// TIA Portal V18 program export: 0 tag tables, 0 data types, 0 data blocks, 2 code blocks (in call order from the OBs), 6 instance data blocks

ORGANIZATION_BLOCK "Main"   // OB1, LAD, ProgramCycle
TITLE = "Main Program Sweep (Cycle)"
{ S7_Optimized_Access := 'TRUE' }
VERSION : 0.1
// Este bloco verifica as condições dos sinais discretos dos painéis. Se as condições operacionais não forem atendidas, as FCs respectivas de cada painel são intertravadas no item 2. Fluxo de Controle.
// stored: AutoNumber true, IsIECCheckEnabled false, SetENOAutomatically false
   VAR_INPUT
      Initial_Call : Bool;   // Initial call of this OB
      Remanence : Bool;   // =True, if remanent data are available
   END_VAR
BEGIN

REGION Network 1: Intertravamento Painel CCO
   // Se o Botão de Emergência estiver Desacionado Painel CCO OK
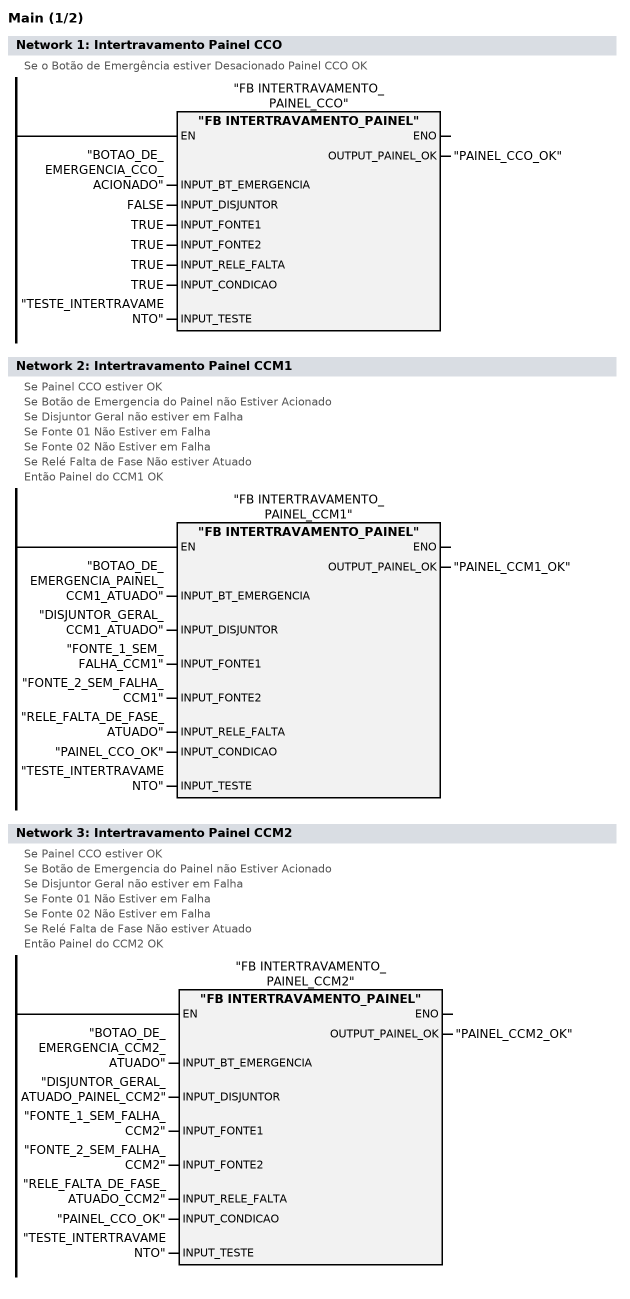
   RUNG wire#powerrail
      "FB INTERTRAVAMENTO_PAINEL_CCO"(INPUT_BT_EMERGENCIA := "BOTAO_DE_EMERGENCIA_CCO_ACIONADO", INPUT_DISJUNTOR := FALSE, INPUT_FONTE1 := TRUE, INPUT_FONTE2 := TRUE, INPUT_RELE_FALTA := TRUE, INPUT_CONDICAO := TRUE, INPUT_TESTE := "TESTE_INTERTRAVAMENTO", OUTPUT_PAINEL_OK => "PAINEL_CCO_OK")
   END_RUNG
   // the same network as SCL:
   "FB INTERTRAVAMENTO_PAINEL_CCO"(INPUT_BT_EMERGENCIA := "BOTAO_DE_EMERGENCIA_CCO_ACIONADO",   // "FB INTERTRAVAMENTO_PAINEL"
                           INPUT_DISJUNTOR := FALSE,
                           INPUT_FONTE1 := TRUE,
                           INPUT_FONTE2 := TRUE,
                           INPUT_RELE_FALTA := TRUE,
                           INPUT_CONDICAO := TRUE,
                           INPUT_TESTE := "TESTE_INTERTRAVAMENTO",
                           OUTPUT_PAINEL_OK => "PAINEL_CCO_OK");
END_REGION

REGION Network 2: Intertravamento Painel CCM1
   // Se Painel CCO estiver OK
   // Se Botão de Emergencia do Painel não Estiver Acionado
   // Se Disjuntor Geral não estiver em Falha
   // Se Fonte 01 Não Estiver em Falha
   // Se Fonte 02 Não Estiver em Falha
   // Se Relé Falta de Fase Não estiver Atuado
   // Então Painel do CCM1 OK
   RUNG wire#powerrail
      "FB INTERTRAVAMENTO_PAINEL_CCM1"(INPUT_BT_EMERGENCIA := "BOTAO_DE_EMERGENCIA_PAINEL_CCM1_ATUADO", INPUT_DISJUNTOR := "DISJUNTOR_GERAL_CCM1_ATUADO", INPUT_FONTE1 := "FONTE_1_SEM_ FALHA_CCM1", INPUT_FONTE2 := "FONTE_2_SEM_FALHA_CCM1", INPUT_RELE_FALTA := "RELE_FALTA_DE_FASE_ATUADO", INPUT_CONDICAO := "PAINEL_CCO_OK", INPUT_TESTE := "TESTE_INTERTRAVAMENTO", OUTPUT_PAINEL_OK => "PAINEL_CCM1_OK")
   END_RUNG
   // the same network as SCL:
   "FB INTERTRAVAMENTO_PAINEL_CCM1"(INPUT_BT_EMERGENCIA := "BOTAO_DE_EMERGENCIA_PAINEL_CCM1_ATUADO",   // "FB INTERTRAVAMENTO_PAINEL"
                           INPUT_DISJUNTOR := "DISJUNTOR_GERAL_CCM1_ATUADO",
                           INPUT_FONTE1 := "FONTE_1_SEM_ FALHA_CCM1",
                           INPUT_FONTE2 := "FONTE_2_SEM_FALHA_CCM1",
                           INPUT_RELE_FALTA := "RELE_FALTA_DE_FASE_ATUADO",
                           INPUT_CONDICAO := "PAINEL_CCO_OK",
                           INPUT_TESTE := "TESTE_INTERTRAVAMENTO",
                           OUTPUT_PAINEL_OK => "PAINEL_CCM1_OK");
END_REGION

REGION Network 3: Intertravamento Painel CCM2
   // Se Painel CCO estiver OK
   // Se Botão de Emergencia do Painel não Estiver Acionado
   // Se Disjuntor Geral não estiver em Falha
   // Se Fonte 01 Não Estiver em Falha
   // Se Fonte 02 Não Estiver em Falha
   // Se Relé Falta de Fase Não estiver Atuado
   // Então Painel do CCM2 OK
   RUNG wire#powerrail
      "FB INTERTRAVAMENTO_PAINEL_CCM2"(INPUT_BT_EMERGENCIA := "BOTAO_DE_EMERGENCIA_CCM2_ATUADO", INPUT_DISJUNTOR := "DISJUNTOR_GERAL_ATUADO_PAINEL_CCM2", INPUT_FONTE1 := "FONTE_1_SEM_FALHA_CCM2", INPUT_FONTE2 := "FONTE_2_SEM_FALHA_CCM2", INPUT_RELE_FALTA := "RELE_FALTA_DE_FASE_ATUADO_CCM2", INPUT_CONDICAO := "PAINEL_CCO_OK", INPUT_TESTE := "TESTE_INTERTRAVAMENTO", OUTPUT_PAINEL_OK => "PAINEL_CCM2_OK")
   END_RUNG
   // the same network as SCL:
   "FB INTERTRAVAMENTO_PAINEL_CCM2"(INPUT_BT_EMERGENCIA := "BOTAO_DE_EMERGENCIA_CCM2_ATUADO",   // "FB INTERTRAVAMENTO_PAINEL"
                           INPUT_DISJUNTOR := "DISJUNTOR_GERAL_ATUADO_PAINEL_CCM2",
                           INPUT_FONTE1 := "FONTE_1_SEM_FALHA_CCM2",
                           INPUT_FONTE2 := "FONTE_2_SEM_FALHA_CCM2",
                           INPUT_RELE_FALTA := "RELE_FALTA_DE_FASE_ATUADO_CCM2",
                           INPUT_CONDICAO := "PAINEL_CCO_OK",
                           INPUT_TESTE := "TESTE_INTERTRAVAMENTO",
                           OUTPUT_PAINEL_OK => "PAINEL_CCM2_OK");
END_REGION

REGION Network 4: Intertravamento Painel CCM3
   // Se Painel CCO estiver OK
   // Se Botão de Emergencia do Painel não Estiver Acionado
   // Se Disjuntor Geral não estiver em Falha
   // Se Fonte 01 Não Estiver em Falha
   // Se Fonte 02 Não Estiver em Falha
   // Se Relé Falta de Fase Não estiver Atuado
   // Então Painel do CCM1 OK
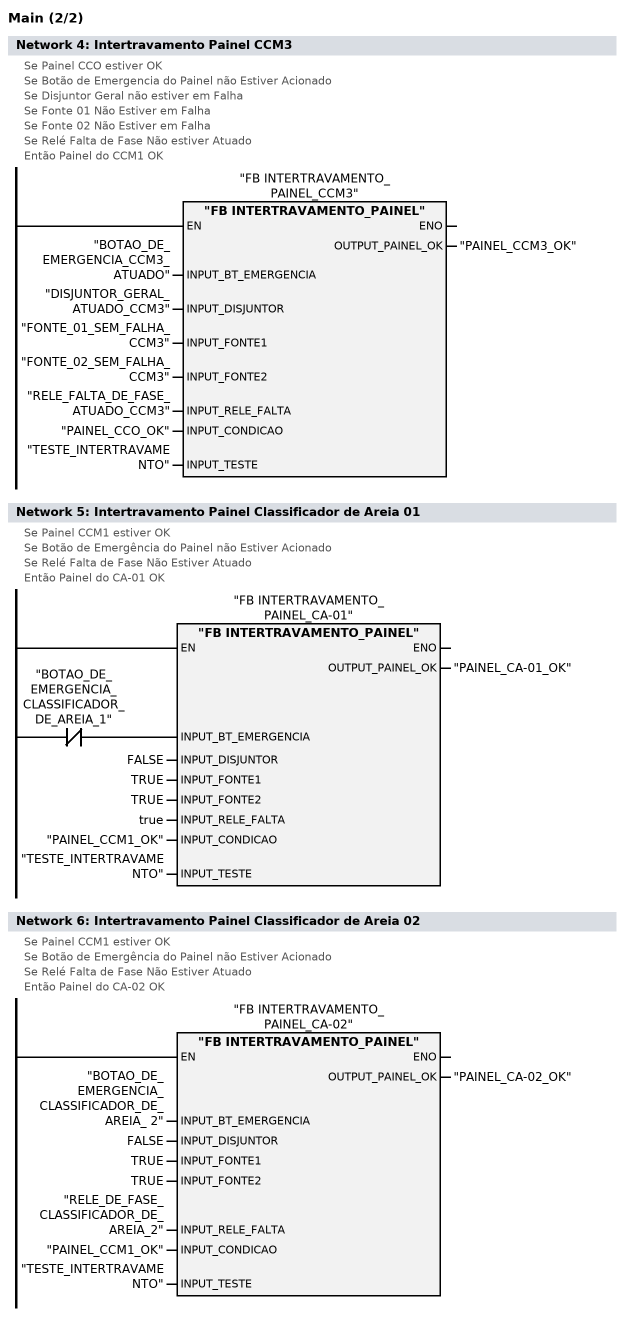
   RUNG wire#powerrail
      "FB INTERTRAVAMENTO_PAINEL_CCM3"(INPUT_BT_EMERGENCIA := "BOTAO_DE_EMERGENCIA_CCM3_ATUADO", INPUT_DISJUNTOR := "DISJUNTOR_GERAL_ATUADO_CCM3", INPUT_FONTE1 := "FONTE_01_SEM_FALHA_CCM3", INPUT_FONTE2 := "FONTE_02_SEM_FALHA_CCM3", INPUT_RELE_FALTA := "RELE_FALTA_DE_FASE_ATUADO_CCM3", INPUT_CONDICAO := "PAINEL_CCO_OK", INPUT_TESTE := "TESTE_INTERTRAVAMENTO", OUTPUT_PAINEL_OK => "PAINEL_CCM3_OK")
   END_RUNG
   // the same network as SCL:
   "FB INTERTRAVAMENTO_PAINEL_CCM3"(INPUT_BT_EMERGENCIA := "BOTAO_DE_EMERGENCIA_CCM3_ATUADO",   // "FB INTERTRAVAMENTO_PAINEL"
                           INPUT_DISJUNTOR := "DISJUNTOR_GERAL_ATUADO_CCM3",
                           INPUT_FONTE1 := "FONTE_01_SEM_FALHA_CCM3",
                           INPUT_FONTE2 := "FONTE_02_SEM_FALHA_CCM3",
                           INPUT_RELE_FALTA := "RELE_FALTA_DE_FASE_ATUADO_CCM3",
                           INPUT_CONDICAO := "PAINEL_CCO_OK",
                           INPUT_TESTE := "TESTE_INTERTRAVAMENTO",
                           OUTPUT_PAINEL_OK => "PAINEL_CCM3_OK");
END_REGION

REGION Network 5: Intertravamento Painel Classificador de Areia 01
   // Se Painel CCM1 estiver OK 
   // Se Botão de Emergência do Painel não Estiver Acionado
   // Se Relé Falta de Fase Não Estiver Atuado 
   // Então Painel do CA-01 OK
   RUNG wire#powerrail
      "FB INTERTRAVAMENTO_PAINEL_CA-01"(INPUT_BT_EMERGENCIA := wire#w1, INPUT_DISJUNTOR := FALSE, INPUT_FONTE1 := TRUE, INPUT_FONTE2 := TRUE, INPUT_RELE_FALTA := true, INPUT_CONDICAO := "PAINEL_CCM1_OK", INPUT_TESTE := "TESTE_INTERTRAVAMENTO", OUTPUT_PAINEL_OK => "PAINEL_CA-01_OK")
   END_RUNG
   RUNG wire#powerrail
      I_Contact( "BOTAO_DE_EMERGENCIA_CLASSIFICADOR_DE_AREIA_1" )
   END_RUNG wire#w1
   // the same network as SCL:
   "FB INTERTRAVAMENTO_PAINEL_CA-01"(INPUT_BT_EMERGENCIA := NOT "BOTAO_DE_EMERGENCIA_CLASSIFICADOR_DE_AREIA_1",   // "FB INTERTRAVAMENTO_PAINEL"
                           INPUT_DISJUNTOR := FALSE,
                           INPUT_FONTE1 := TRUE,
                           INPUT_FONTE2 := TRUE,
                           INPUT_RELE_FALTA := true,
                           INPUT_CONDICAO := "PAINEL_CCM1_OK",
                           INPUT_TESTE := "TESTE_INTERTRAVAMENTO",
                           OUTPUT_PAINEL_OK => "PAINEL_CA-01_OK");
END_REGION

REGION Network 6: Intertravamento Painel Classificador de Areia 02
   // Se Painel CCM1 estiver OK 
   // Se Botão de Emergência do Painel não Estiver Acionado
   // Se Relé Falta de Fase Não Estiver Atuado 
   // Então Painel do CA-02 OK
   RUNG wire#powerrail
      "FB INTERTRAVAMENTO_PAINEL_CA-02"(INPUT_BT_EMERGENCIA := "BOTAO_DE_EMERGENCIA_CLASSIFICADOR_DE_AREIA_ 2", INPUT_DISJUNTOR := FALSE, INPUT_FONTE1 := TRUE, INPUT_FONTE2 := TRUE, INPUT_RELE_FALTA := "RELE_DE_FASE_CLASSIFICADOR_DE_AREIA_2", INPUT_CONDICAO := "PAINEL_CCM1_OK", INPUT_TESTE := "TESTE_INTERTRAVAMENTO", OUTPUT_PAINEL_OK => "PAINEL_CA-02_OK")
   END_RUNG
   // the same network as SCL:
   "FB INTERTRAVAMENTO_PAINEL_CA-02"(INPUT_BT_EMERGENCIA := "BOTAO_DE_EMERGENCIA_CLASSIFICADOR_DE_AREIA_ 2",   // "FB INTERTRAVAMENTO_PAINEL"
                           INPUT_DISJUNTOR := FALSE,
                           INPUT_FONTE1 := TRUE,
                           INPUT_FONTE2 := TRUE,
                           INPUT_RELE_FALTA := "RELE_DE_FASE_CLASSIFICADOR_DE_AREIA_2",
                           INPUT_CONDICAO := "PAINEL_CCM1_OK",
                           INPUT_TESTE := "TESTE_INTERTRAVAMENTO",
                           OUTPUT_PAINEL_OK => "PAINEL_CA-02_OK");
END_REGION

REGION Network 7: Comunicação Supervisório
END_REGION
END_ORGANIZATION_BLOCK

ORGANIZATION_BLOCK "Resets"   // OB126, LAD, ProgramCycle
TITLE = "Main Program Sweep (Cycle)"
{ S7_Optimized_Access := 'TRUE' }
VERSION : 0.1
// stored: AutoNumber true, IsIECCheckEnabled false, SetENOAutomatically false
   VAR_INPUT
      Initial_Call : Bool;   // Initial call of this OB
      Remanence : Bool;   // =True, if remanent data are available
   END_VAR
   VAR_TEMP   // added for the SCL form of the ladder/FBD networks
      _w1 : Bool;
   END_VAR
BEGIN

REGION Network 1: Reset Aferição (Inversor/Instrumentação)
   // Se o valor do comando de aferição for diferente de 0, um tempo será disparado para que a aferição seja feita, em seguida, os valores de entrada serão zerados
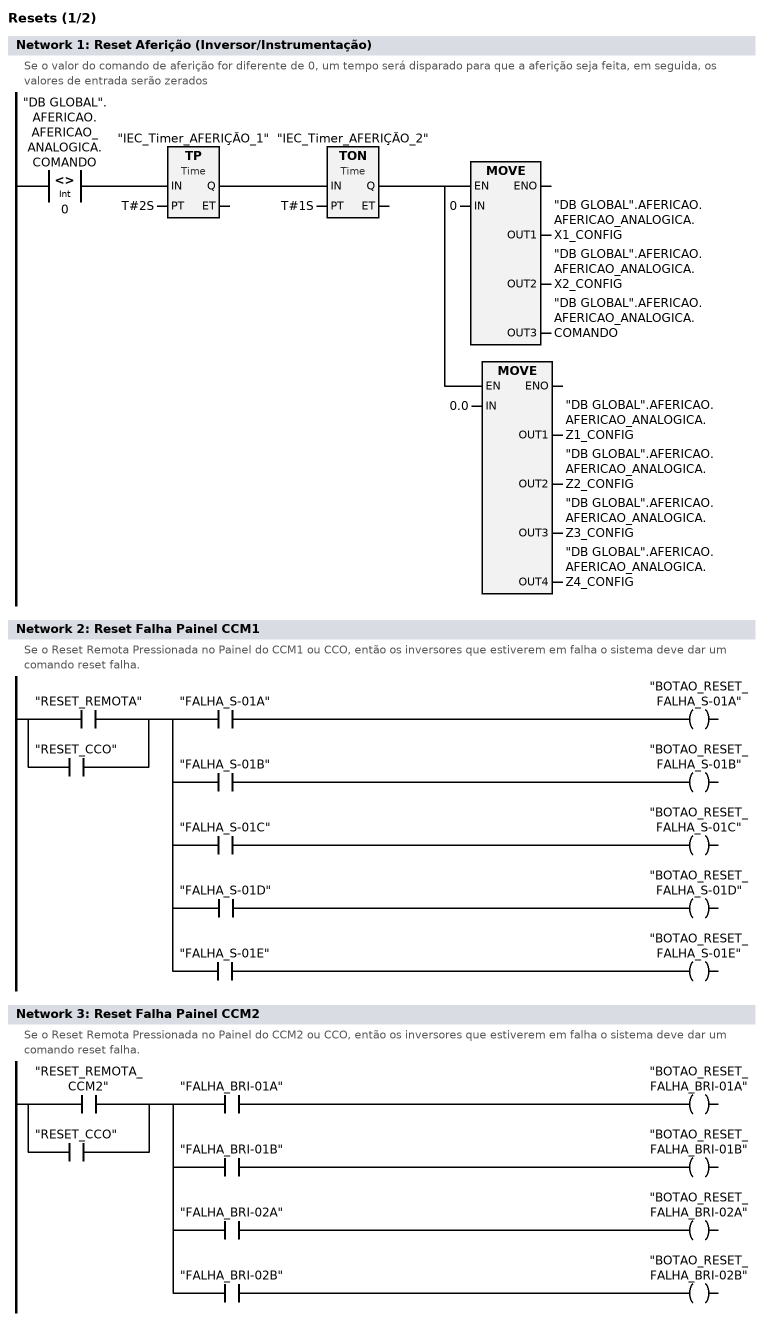
   RUNG wire#powerrail
      { S7_Templates := "SrcType := Int" } NE_Contact(in1 := "DB GLOBAL".AFERICAO.AFERICAO_ANALOGICA.COMANDO, in2 := 0)
      { S7_Templates := "time_type := Time" } "IEC_Timer_AFERIÇÃO_1".TP(pt := T#2S, et =>)
      { S7_Templates := "time_type := Time" } "IEC_Timer_AFERIÇÃO_2".TON(pt := T#1S, et =>)
      wire#w1
      Move(in := 0, out1 => "DB GLOBAL".AFERICAO.AFERICAO_ANALOGICA.X1_CONFIG, out2 => "DB GLOBAL".AFERICAO.AFERICAO_ANALOGICA.X2_CONFIG, out3 => "DB GLOBAL".AFERICAO.AFERICAO_ANALOGICA.COMANDO)
   END_RUNG
   RUNG wire#w1
      Move(in := 0.0, out1 => "DB GLOBAL".AFERICAO.AFERICAO_ANALOGICA.Z1_CONFIG, out2 => "DB GLOBAL".AFERICAO.AFERICAO_ANALOGICA.Z2_CONFIG, out3 => "DB GLOBAL".AFERICAO.AFERICAO_ANALOGICA.Z3_CONFIG, out4 => "DB GLOBAL".AFERICAO.AFERICAO_ANALOGICA.Z4_CONFIG)
   END_RUNG
   // the same network as SCL:
   "IEC_Timer_AFERIÇÃO_1".TP(IN := "DB GLOBAL".AFERICAO.AFERICAO_ANALOGICA.COMANDO <> 0, PT := T#2S);
   "IEC_Timer_AFERIÇÃO_2".TON(IN := "IEC_Timer_AFERIÇÃO_1".Q, PT := T#1S);
   IF "IEC_Timer_AFERIÇÃO_2".Q THEN
       "DB GLOBAL".AFERICAO.AFERICAO_ANALOGICA.X1_CONFIG := 0;
       "DB GLOBAL".AFERICAO.AFERICAO_ANALOGICA.X2_CONFIG := 0;
       "DB GLOBAL".AFERICAO.AFERICAO_ANALOGICA.COMANDO := 0;
       "DB GLOBAL".AFERICAO.AFERICAO_ANALOGICA.Z1_CONFIG := 0.0;
       "DB GLOBAL".AFERICAO.AFERICAO_ANALOGICA.Z2_CONFIG := 0.0;
       "DB GLOBAL".AFERICAO.AFERICAO_ANALOGICA.Z3_CONFIG := 0.0;
       "DB GLOBAL".AFERICAO.AFERICAO_ANALOGICA.Z4_CONFIG := 0.0;
   END_IF;
END_REGION

REGION Network 2: Reset Falha Painel CCM1
   // Se o Reset Remota Pressionada no Painel do CCM1 ou CCO, então os inversores que estiverem em falha o sistema deve dar um comando reset falha.
   RUNG wire#powerrail
      Contact( "RESET_REMOTA" )
      wire#w1
      Contact( "FALHA_S-01A" )
      Coil( "BOTAO_RESET_FALHA_S-01A" )
   END_RUNG
   RUNG wire#powerrail
      Contact( "RESET_CCO" )
   END_RUNG wire#w1
   RUNG wire#w1
      Contact( "FALHA_S-01B" )
      Coil( "BOTAO_RESET_FALHA_S-01B" )
   END_RUNG
   RUNG wire#w1
      Contact( "FALHA_S-01C" )
      Coil( "BOTAO_RESET_FALHA_S-01C" )
   END_RUNG
   RUNG wire#w1
      Contact( "FALHA_S-01D" )
      Coil( "BOTAO_RESET_FALHA_S-01D" )
   END_RUNG
   RUNG wire#w1
      Contact( "FALHA_S-01E" )
      Coil( "BOTAO_RESET_FALHA_S-01E" )
   END_RUNG
   // the same network as SCL:
   #_w1 := "RESET_REMOTA" OR "RESET_CCO";
   "BOTAO_RESET_FALHA_S-01A" := #_w1 AND "FALHA_S-01A";
   "BOTAO_RESET_FALHA_S-01B" := #_w1 AND "FALHA_S-01B";
   "BOTAO_RESET_FALHA_S-01C" := #_w1 AND "FALHA_S-01C";
   "BOTAO_RESET_FALHA_S-01D" := #_w1 AND "FALHA_S-01D";
   "BOTAO_RESET_FALHA_S-01E" := #_w1 AND "FALHA_S-01E";
END_REGION

REGION Network 3: Reset Falha Painel CCM2
   // Se o Reset Remota Pressionada no Painel do CCM2 ou CCO, então os inversores que estiverem em falha o sistema deve dar um comando reset falha.
   RUNG wire#powerrail
      Contact( "RESET_REMOTA_CCM2" )
      wire#w1
      Contact( "FALHA_BRI-01A" )
      Coil( "BOTAO_RESET_FALHA_BRI-01A" )
   END_RUNG
   RUNG wire#powerrail
      Contact( "RESET_CCO" )
   END_RUNG wire#w1
   RUNG wire#w1
      Contact( "FALHA_BRI-01B" )
      Coil( "BOTAO_RESET_FALHA_BRI-01B" )
   END_RUNG
   RUNG wire#w1
      Contact( "FALHA_BRI-02A" )
      Coil( "BOTAO_RESET_FALHA_BRI-02A" )
   END_RUNG
   RUNG wire#w1
      Contact( "FALHA_BRI-02B" )
      Coil( "BOTAO_RESET_FALHA_BRI-02B" )
   END_RUNG
   // the same network as SCL:
   #_w1 := "RESET_REMOTA_CCM2" OR "RESET_CCO";
   "BOTAO_RESET_FALHA_BRI-01A" := #_w1 AND "FALHA_BRI-01A";
   "BOTAO_RESET_FALHA_BRI-01B" := #_w1 AND "FALHA_BRI-01B";
   "BOTAO_RESET_FALHA_BRI-02A" := #_w1 AND "FALHA_BRI-02A";
   "BOTAO_RESET_FALHA_BRI-02B" := #_w1 AND "FALHA_BRI-02B";
END_REGION

REGION Network 4: Reset Reset Painel CCM3
   // Se o Reset Remota Pressionada no Painel do CCM3 ou CCO, então os inversores que estiverem em falha o sistema deve dar um comando reset falha.
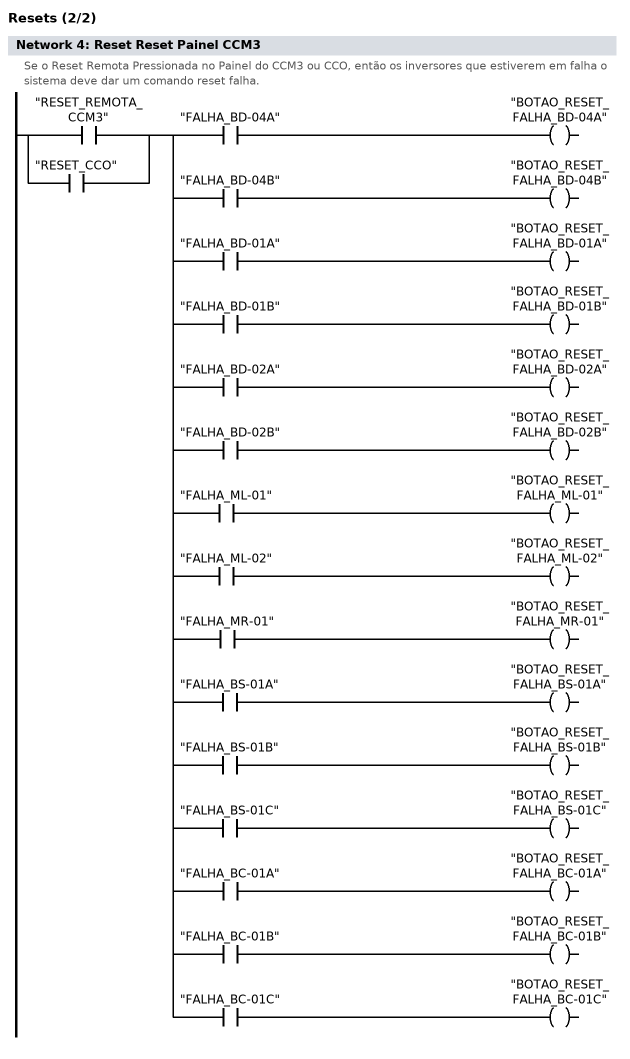
   RUNG wire#powerrail
      Contact( "RESET_REMOTA_CCM3" )
      wire#w1
      Contact( "FALHA_BD-04A" )
      Coil( "BOTAO_RESET_FALHA_BD-04A" )
   END_RUNG
   RUNG wire#powerrail
      Contact( "RESET_CCO" )
   END_RUNG wire#w1
   RUNG wire#w1
      Contact( "FALHA_BD-04B" )
      Coil( "BOTAO_RESET_FALHA_BD-04B" )
   END_RUNG
   RUNG wire#w1
      Contact( "FALHA_BD-01A" )
      Coil( "BOTAO_RESET_FALHA_BD-01A" )
   END_RUNG
   RUNG wire#w1
      Contact( "FALHA_BD-01B" )
      Coil( "BOTAO_RESET_FALHA_BD-01B" )
   END_RUNG
   RUNG wire#w1
      Contact( "FALHA_BD-02A" )
      Coil( "BOTAO_RESET_FALHA_BD-02A" )
   END_RUNG
   RUNG wire#w1
      Contact( "FALHA_BD-02B" )
      Coil( "BOTAO_RESET_FALHA_BD-02B" )
   END_RUNG
   RUNG wire#w1
      Contact( "FALHA_ML-01" )
      Coil( "BOTAO_RESET_FALHA_ML-01" )
   END_RUNG
   RUNG wire#w1
      Contact( "FALHA_ML-02" )
      Coil( "BOTAO_RESET_FALHA_ML-02" )
   END_RUNG
   RUNG wire#w1
      Contact( "FALHA_MR-01" )
      Coil( "BOTAO_RESET_FALHA_MR-01" )
   END_RUNG
   RUNG wire#w1
      Contact( "FALHA_BS-01A" )
      Coil( "BOTAO_RESET_FALHA_BS-01A" )
   END_RUNG
   RUNG wire#w1
      Contact( "FALHA_BS-01B" )
      Coil( "BOTAO_RESET_FALHA_BS-01B" )
   END_RUNG
   RUNG wire#w1
      Contact( "FALHA_BS-01C" )
      Coil( "BOTAO_RESET_FALHA_BS-01C" )
   END_RUNG
   RUNG wire#w1
      Contact( "FALHA_BC-01A" )
      Coil( "BOTAO_RESET_FALHA_BC-01A" )
   END_RUNG
   RUNG wire#w1
      Contact( "FALHA_BC-01B" )
      Coil( "BOTAO_RESET_FALHA_BC-01B" )
   END_RUNG
   RUNG wire#w1
      Contact( "FALHA_BC-01C" )
      Coil( "BOTAO_RESET_FALHA_BC-01C" )
   END_RUNG
   // the same network as SCL:
   #_w1 := "RESET_REMOTA_CCM3" OR "RESET_CCO";
   "BOTAO_RESET_FALHA_BD-04A" := #_w1 AND "FALHA_BD-04A";
   "BOTAO_RESET_FALHA_BD-04B" := #_w1 AND "FALHA_BD-04B";
   "BOTAO_RESET_FALHA_BD-01A" := #_w1 AND "FALHA_BD-01A";
   "BOTAO_RESET_FALHA_BD-01B" := #_w1 AND "FALHA_BD-01B";
   "BOTAO_RESET_FALHA_BD-02A" := #_w1 AND "FALHA_BD-02A";
   "BOTAO_RESET_FALHA_BD-02B" := #_w1 AND "FALHA_BD-02B";
   "BOTAO_RESET_FALHA_ML-01" := #_w1 AND "FALHA_ML-01";
   "BOTAO_RESET_FALHA_ML-02" := #_w1 AND "FALHA_ML-02";
   "BOTAO_RESET_FALHA_MR-01" := #_w1 AND "FALHA_MR-01";
   "BOTAO_RESET_FALHA_BS-01A" := #_w1 AND "FALHA_BS-01A";
   "BOTAO_RESET_FALHA_BS-01B" := #_w1 AND "FALHA_BS-01B";
   "BOTAO_RESET_FALHA_BS-01C" := #_w1 AND "FALHA_BS-01C";
   "BOTAO_RESET_FALHA_BC-01A" := #_w1 AND "FALHA_BC-01A";
   "BOTAO_RESET_FALHA_BC-01B" := #_w1 AND "FALHA_BC-01B";
   "BOTAO_RESET_FALHA_BC-01C" := #_w1 AND "FALHA_BC-01C";
END_REGION
END_ORGANIZATION_BLOCK

DATA_BLOCK "FB INTERTRAVAMENTO_PAINEL_CA-01"   // DB597
VERSION : 0.1
// stored: AutoNumber true, DBAccessibleFromOPCUA true, DBAccessibleFromWebserver true, InstanceOfName FB INTERTRAVAMENTO_PAINEL, InstanceOfType FB
"FB INTERTRAVAMENTO_PAINEL"
   // VAR_INPUT
   //    INPUT_BT_EMERGENCIA : Bool;
   //    INPUT_DISJUNTOR : Bool;
   //    INPUT_FONTE1 : Bool;
   //    INPUT_FONTE2 : Bool;
   //    INPUT_RELE_FALTA : Bool;
   //    INPUT_CONDICAO : Bool;
   //    INPUT_TESTE : Bool;
   // END_VAR
   // VAR_OUTPUT
   //    OUTPUT_PAINEL_OK : Bool;
   // END_VAR
BEGIN
END_DATA_BLOCK

DATA_BLOCK "FB INTERTRAVAMENTO_PAINEL_CA-02"   // DB598
VERSION : 0.1
// stored: AutoNumber true, DBAccessibleFromOPCUA true, DBAccessibleFromWebserver true, InstanceOfName FB INTERTRAVAMENTO_PAINEL, InstanceOfType FB
"FB INTERTRAVAMENTO_PAINEL"
   // VAR_INPUT
   //    INPUT_BT_EMERGENCIA : Bool;
   //    INPUT_DISJUNTOR : Bool;
   //    INPUT_FONTE1 : Bool;
   //    INPUT_FONTE2 : Bool;
   //    INPUT_RELE_FALTA : Bool;
   //    INPUT_CONDICAO : Bool;
   //    INPUT_TESTE : Bool;
   // END_VAR
   // VAR_OUTPUT
   //    OUTPUT_PAINEL_OK : Bool;
   // END_VAR
BEGIN
END_DATA_BLOCK

DATA_BLOCK "FB INTERTRAVAMENTO_PAINEL_CCM1"   // DB594
VERSION : 0.1
// stored: AutoNumber true, DBAccessibleFromOPCUA true, DBAccessibleFromWebserver true, InstanceOfName FB INTERTRAVAMENTO_PAINEL, InstanceOfType FB
"FB INTERTRAVAMENTO_PAINEL"
   // VAR_INPUT
   //    INPUT_BT_EMERGENCIA : Bool;
   //    INPUT_DISJUNTOR : Bool;
   //    INPUT_FONTE1 : Bool;
   //    INPUT_FONTE2 : Bool;
   //    INPUT_RELE_FALTA : Bool;
   //    INPUT_CONDICAO : Bool;
   //    INPUT_TESTE : Bool;
   // END_VAR
   // VAR_OUTPUT
   //    OUTPUT_PAINEL_OK : Bool;
   // END_VAR
BEGIN
END_DATA_BLOCK

DATA_BLOCK "FB INTERTRAVAMENTO_PAINEL_CCM2"   // DB595
VERSION : 0.1
// stored: AutoNumber true, DBAccessibleFromOPCUA true, DBAccessibleFromWebserver true, InstanceOfName FB INTERTRAVAMENTO_PAINEL, InstanceOfType FB
"FB INTERTRAVAMENTO_PAINEL"
   // VAR_INPUT
   //    INPUT_BT_EMERGENCIA : Bool;
   //    INPUT_DISJUNTOR : Bool;
   //    INPUT_FONTE1 : Bool;
   //    INPUT_FONTE2 : Bool;
   //    INPUT_RELE_FALTA : Bool;
   //    INPUT_CONDICAO : Bool;
   //    INPUT_TESTE : Bool;
   // END_VAR
   // VAR_OUTPUT
   //    OUTPUT_PAINEL_OK : Bool;
   // END_VAR
BEGIN
END_DATA_BLOCK

DATA_BLOCK "FB INTERTRAVAMENTO_PAINEL_CCM3"   // DB596
VERSION : 0.1
// stored: AutoNumber true, DBAccessibleFromOPCUA true, DBAccessibleFromWebserver true, InstanceOfName FB INTERTRAVAMENTO_PAINEL, InstanceOfType FB
"FB INTERTRAVAMENTO_PAINEL"
   // VAR_INPUT
   //    INPUT_BT_EMERGENCIA : Bool;
   //    INPUT_DISJUNTOR : Bool;
   //    INPUT_FONTE1 : Bool;
   //    INPUT_FONTE2 : Bool;
   //    INPUT_RELE_FALTA : Bool;
   //    INPUT_CONDICAO : Bool;
   //    INPUT_TESTE : Bool;
   // END_VAR
   // VAR_OUTPUT
   //    OUTPUT_PAINEL_OK : Bool;
   // END_VAR
BEGIN
END_DATA_BLOCK

DATA_BLOCK "FB INTERTRAVAMENTO_PAINEL_CCO"   // DB599
VERSION : 0.1
// stored: AutoNumber true, DBAccessibleFromOPCUA true, DBAccessibleFromWebserver true, InstanceOfName FB INTERTRAVAMENTO_PAINEL, InstanceOfType FB
"FB INTERTRAVAMENTO_PAINEL"
   // VAR_INPUT
   //    INPUT_BT_EMERGENCIA : Bool;
   //    INPUT_DISJUNTOR : Bool;
   //    INPUT_FONTE1 : Bool;
   //    INPUT_FONTE2 : Bool;
   //    INPUT_RELE_FALTA : Bool;
   //    INPUT_CONDICAO : Bool;
   //    INPUT_TESTE : Bool;
   // END_VAR
   // VAR_OUTPUT
   //    OUTPUT_PAINEL_OK : Bool;
   // END_VAR
BEGIN
END_DATA_BLOCK
